FUNCTION_BLOCK E_MUX8 (* Event multiplexer 8 Events *)
  (* Standard: 61499-1 Annex A; Description: Copyright (c) 2017, 2025 fortiss GmbH, HR Agrartechnik GmbH This program and the accompanying materials are made available under the terms of the Eclipse Public License 2.0 which is available at https://www.eclipse.org/legal/epl-2.0/ SPDX-License-Identifier: EPL-2.0 *)
  (* Version 1.0, 2017-09-22, Alois Zoitl, fortiss GmbH, initial API and implementation and/or initial documentation *)
  (* Version 1.1, 2025-02-16, Franz Höpfinger, HR Agrartechnik GmbH, Copy E_DEMUX8 and made E_MUX8 *)
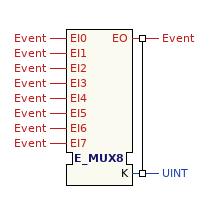
  EVENT_INPUT
    EI0;
    EI1;
    EI2;
    EI3;
    EI4;
    EI5;
    EI6;
    EI7;
  END_EVENT
  EVENT_OUTPUT
    EO WITH K; (* Event which was multiplexed *)
  END_EVENT
  VAR_OUTPUT
    K : UINT; (* Event index *)
  END_VAR
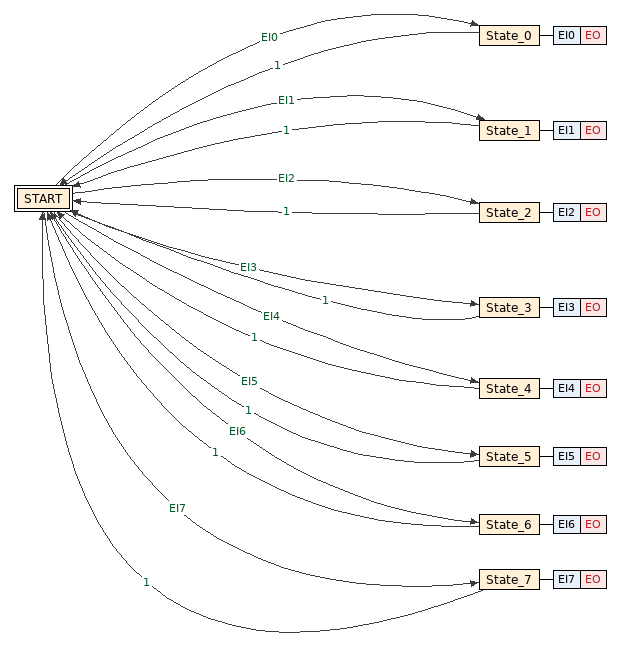
  EC_STATES
    START; (* Initial State *)
    State_0 : EI0 -> EO;
    State_1 : EI1 -> EO;
    State_2 : EI2 -> EO;
    State_3 : EI3 -> EO;
    State_4 : EI4 -> EO;
    State_5 : EI5 -> EO;
    State_6 : EI6 -> EO;
    State_7 : EI7 -> EO;
  END_STATES
  EC_TRANSITIONS
    State_0 TO START := 1;
    State_1 TO START := 1;
    State_2 TO START := 1;
    State_3 TO START := 1;
    START TO State_0 := EI0;
    START TO State_1 := EI1;
    START TO State_2 := EI2;
    START TO State_3 := EI3;
    State_4 TO START := 1;
    State_5 TO START := 1;
    State_6 TO START := 1;
    State_7 TO START := 1;
    START TO State_4 := EI4;
    START TO State_5 := EI5;
    START TO State_6 := EI6;
    START TO State_7 := EI7;
  END_TRANSITIONS
  ALGORITHM EI0 IN ST:
K := 0;
  END_ALGORITHM
  ALGORITHM EI1 IN ST:
K := 1;
  END_ALGORITHM
  ALGORITHM EI2 IN ST:
K := 2;
  END_ALGORITHM
  ALGORITHM EI3 IN ST:
K := 3;
  END_ALGORITHM
  ALGORITHM EI4 IN ST:
K := 4;
  END_ALGORITHM
  ALGORITHM EI5 IN ST:
K := 5;
  END_ALGORITHM
  ALGORITHM EI6 IN ST:
K := 6;
  END_ALGORITHM
  ALGORITHM EI7 IN ST:
K := 7;
  END_ALGORITHM
END_FUNCTION_BLOCK
